{attribute 'qualified_only'}
{attribute 'strict'}
TYPE E_CheckFileExistsStates :
(	
	WaitForStart,
	WaitForOpenResult,
	CloseIfOpened
);
END_TYPE

(* stored: Version 1.1.0.1, ProductVersion 3.1.4022.18
   DUT E_CheckFileExistsStates: Id {2d38e022-fe51-08c3-2bd2-65303a03174c} *)
